// Mitsubishi GX Works2 project: ex2 (1) (1)   PLC: FX3G

// global labels: Global1
VAR_GLOBAL CONSTANT
  cream_dose : INT := 300;
  chocolate_dose : INT := 120;
END_VAR
VAR_GLOBAL
  Analog_Input AT D8280 : INT;
  Analog_Input1 AT D8201 : INT;
  SYSTEM AT M0 : BOOL;
  Y_1 AT Y001 : BOOL;
  Y_0 AT Y000 : BOOL;
  IsCocolate AT M0 : BOOL;
  CreamIsOver AT M4 : BOOL;
  CocolateIsOver AT M3 : BOOL;
  DoubelChocolate AT D1111 : INT;
  UseChocolate AT D8203 : INT;
  CreamFlickering AT CC3 : BOOL;
  SCreamFlickering AT CS3 : BOOL;
  CreamTimer1 AT TC3 : BOOL;
  CreamTimer2 AT TC4 : BOOL;
  SCreamTimer1 AT TS3 : BOOL;
  SCreamTimer2 AT TS4 : BOOL;
  SystemStart AT X007 : BOOL;
  SystemON AT M10 : BOOL;
  SEndFlickering AT CS1 : BOOL;
  EndFlickering AT CC1 : BOOL;
  EndTimer1 AT TC1 : BOOL;
  EndTimer2 AT TC2 : BOOL;
  SEndTimer1 AT TS1 : BOOL;
  SEndFlickering1 AT TS1 : BOOL;
END_VAR
VAR_GLOBAL CONSTANT
  K_5 : INT := 5;
  K_8 : INT := 8;
  k_0 : INT;
  K_4 : INT := 4;
  K_6 : INT := 6;
  K_10 : INT := 10;
END_VAR
VAR_GLOBAL
  EddChocolate AT X006 : BOOL;
  EddCream AT X011 : BOOL;
  UseCream AT D8205 : INT;
END_VAR
VAR_GLOBAL CONSTANT
  K_3 : INT := 3;
END_VAR
VAR_GLOBAL
  Y_3 AT Y003 : BOOL;
  CocolateTimer1 AT TC8 : BOOL;
  CocolateTimer1OUT AT TS8 : BOOL;
END_VAR
VAR_GLOBAL CONSTANT
  K_50 : INT := 50;
  K_6V : INT := 2340;
END_VAR
VAR_GLOBAL
  SEndTimer2 AT TS2 : BOOL;
  Y_007 AT Y007 : BOOL;
  cream_stock AT D8230 : INT;
  chocolate_stock AT D8232 : INT;
  Pack AT X000 : BOOL;
  CC10 AT CC10 : BOOL;
  Packing AT X000 : BOOL;
  Packing2 AT Y002 : BOOL;
  nomberOfKrembo AT CC11 : BOOL;
END_VAR
VAR_GLOBAL CONSTANT
  K_3200 : INT := 3200;
END_VAR
VAR_GLOBAL
  NnomberOfKrembo AT CN11 : INT;
  Finished AT D8210 : INT;
  Finished_pack AT CC12 : BOOL;
  NFinishedPack AT CN12 : INT;
END_VAR

// task Task_01 (event TRUE, interval 0, priority 31): POU_01

PROGRAM POU_01
(* structured ladder/FBD written out as ST: instructions are called as NAME(EN, inputs, outputs); _pN, _eN, _tN stand for wires *)
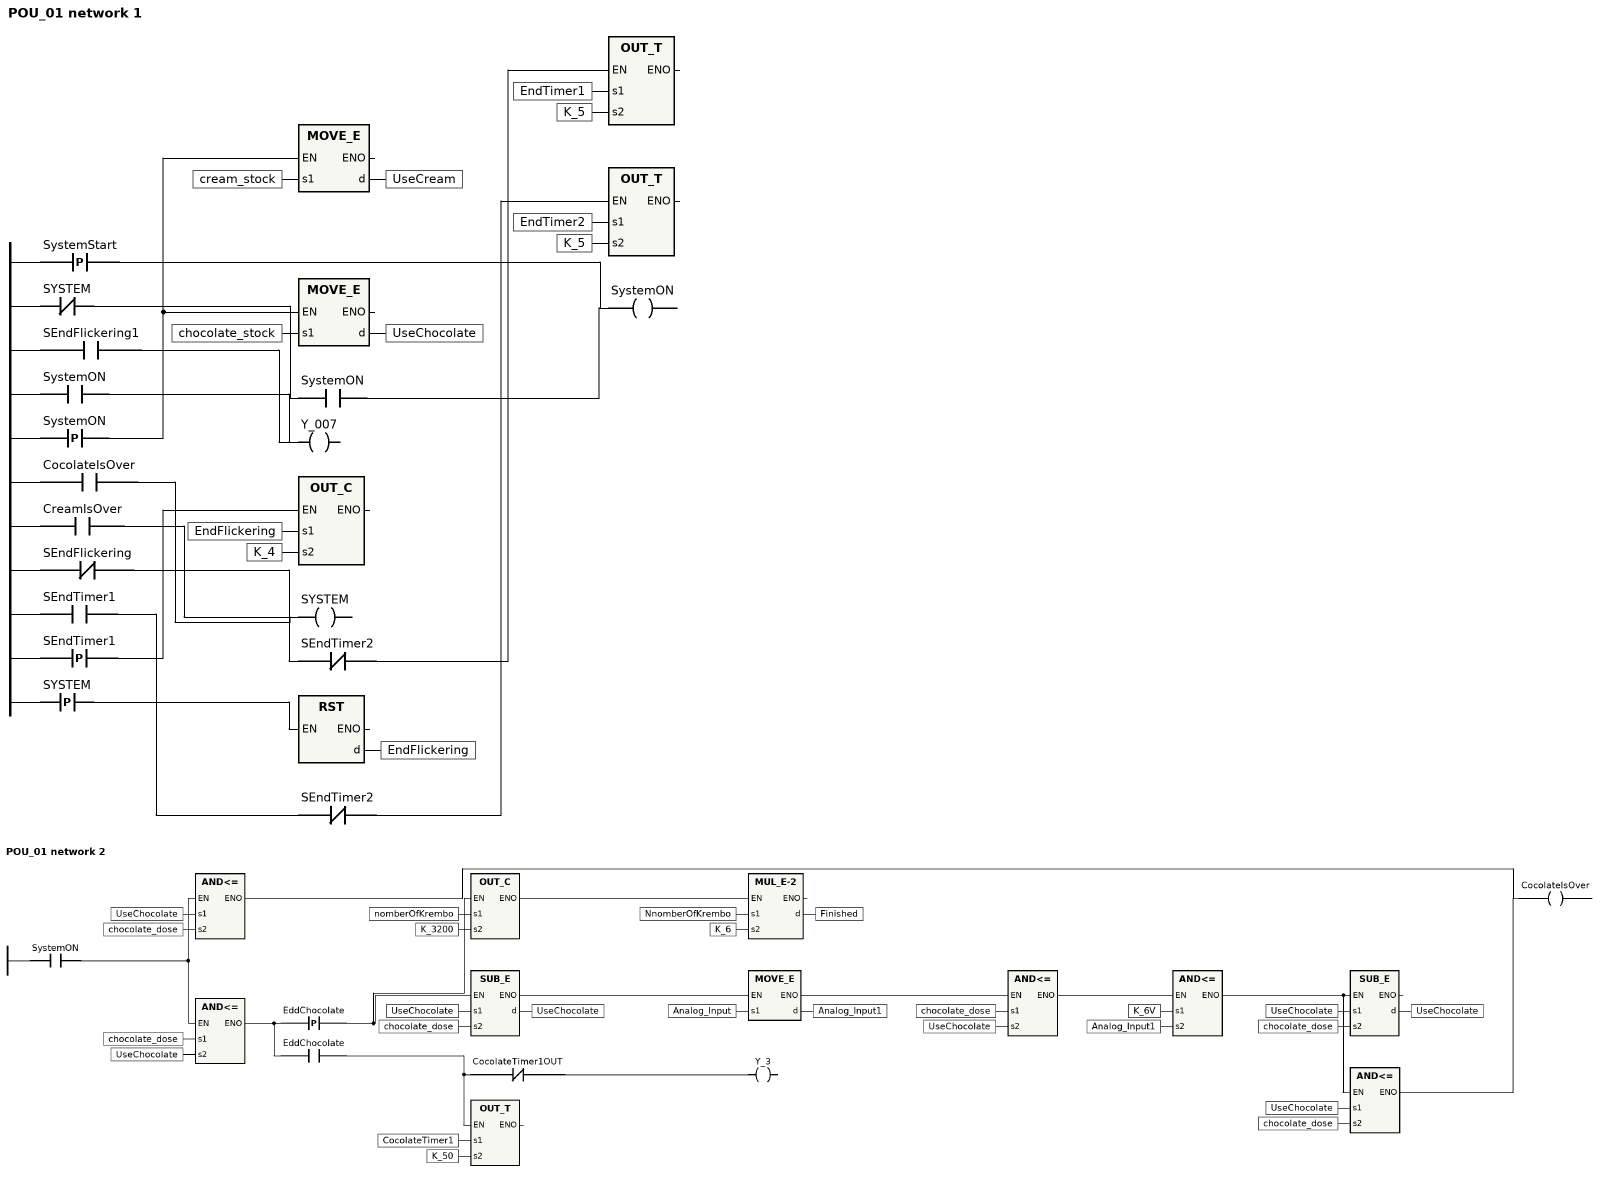
(* network 1 *)
SystemON := LDP(TRUE, SystemStart) OR (NOT SYSTEM AND SystemON);
Y_007 := SEndFlickering1 OR SystemON;
_p1 := LDP(TRUE, SystemON);
MOVE_E(_p1, cream_stock, UseCream);
MOVE_E(_p1, chocolate_stock, UseChocolate);
SYSTEM := CocolateIsOver OR CreamIsOver;
OUT_T(NOT SEndFlickering AND NOT SEndTimer2, EndTimer1, K_5);
OUT_T(SEndTimer1 AND NOT SEndTimer2, EndTimer2, K_5);
OUT_C(LDP(TRUE, SEndTimer1), EndFlickering, K_4);
RST(LDP(TRUE, SYSTEM), EndFlickering);
(* network 2 *)
_e1 := AND<=(SystemON, UseChocolate, chocolate_dose);
_e2 := AND<=(SystemON, chocolate_dose, UseChocolate);
_p3 := _e2 AND LDP(TRUE, EddChocolate);
_e4 := OUT_C(_p3, nomberOfKrembo, K_3200);
MUL_E(_e4, NnomberOfKrembo, K_6, Finished);
_e5 := SUB_E(_p3, UseChocolate, chocolate_dose, UseChocolate);
_e6 := MOVE_E(_e5, Analog_Input, Analog_Input1);
_e7 := AND<=(_e6, chocolate_dose, UseChocolate);
_e8 := AND<=(_e7, K_6V, Analog_Input1);
_e9 := AND<=(_e8, UseChocolate, chocolate_dose);
CocolateIsOver := _e1 OR _e9;
SUB_E(_e8, UseChocolate, chocolate_dose, UseChocolate);
_p10 := _e2 AND EddChocolate;
OUT_T(_p10, CocolateTimer1, K_50);
Y_3 := _p10 AND NOT CocolateTimer1OUT;
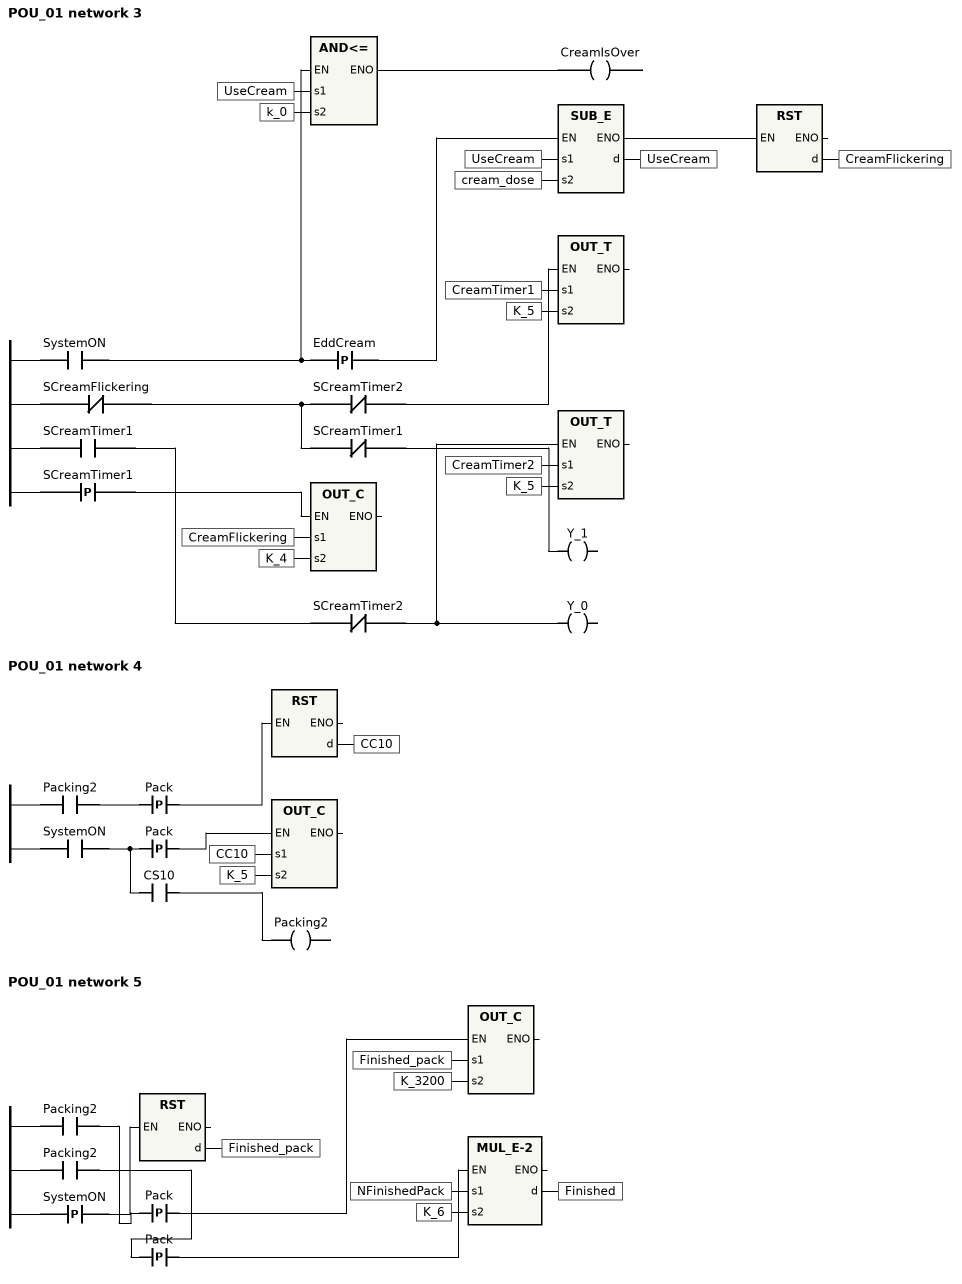
(* network 3 *)
_e1 := AND<=(SystemON, UseCream, k_0);
CreamIsOver := _e1;
_e2 := SUB_E(SystemON AND LDP(TRUE, EddCream), UseCream, cream_dose, UseCream);
RST(_e2, CreamFlickering);
_p3 := NOT SCreamFlickering;
OUT_T(_p3 AND NOT SCreamTimer2, CreamTimer1, K_5);
Y_1 := _p3 AND NOT SCreamTimer1;
_p4 := SCreamTimer1 AND NOT SCreamTimer2;
OUT_T(_p4, CreamTimer2, K_5);
Y_0 := _p4;
OUT_C(LDP(TRUE, SCreamTimer1), CreamFlickering, K_4);
(* network 4 *)
RST(Packing2 AND LDP(TRUE, Pack), CC10);
OUT_C(SystemON AND LDP(TRUE, Pack), CC10, K_5);
Packing2 := SystemON AND CS10;
(* network 5 *)
OUT_C(Packing2 AND LDP(TRUE, Pack), Finished_pack, K_3200);
MUL_E(Packing2 AND LDP(TRUE, Pack), NFinishedPack, K_6, Finished);
RST(LDP(TRUE, SystemON), Finished_pack);
END_PROGRAM
